Staubli VAL3: markItem.pgx

public program markItem(num x_nIndex, string x_sName)
begin
  if left(sml:box[x_sName].comment[x_nIndex],1)!="#"
    sml:box[x_sName].comment[x_nIndex]="# "+sml:box[x_sName].comment[x_nIndex]
  else
    sml:box[x_sName].comment[x_nIndex]=right(sml:box[x_sName].comment[x_nIndex],len(sml:box[x_sName].comment[x_nIndex])-2)
  endIf
end
